// TIA Portal V17 export
// export: Created 2022-03-12T16:05:29.6133544Z, ExportSetting WithDefaults, DisplayName Totally Integrated Automation Portal, DisplayVersion V17, DisplayName TIA Portal Openness, DisplayVersion V17, DisplayName TIA Portal Version Control Interface, DisplayVersion V17, DisplayName STEP 7 Professional, DisplayVersion V17, DisplayName STEP 7 Safety, DisplayVersion V17, DisplayName WinCC Advanced / Unified PC, DisplayVersion V17
DATA_BLOCK "StatusCfg"   // DB31602
TITLE = CPG_StatusCfg
{ S7_Optimized_Access := 'TRUE' }
AUTHOR : tech.team.motioncontrol@siemens.com
FAMILY : CPG
VERSION : 1.0
// Support: tech.team.motioncontrol@siemens.com
// Fax: +49 (0) 9131/98-1297
// stored: AutoNumber true, DBAccessibleFromOPCUA true, DBAccessibleFromWebserver true, IsOnlyStoredInLoadMemory false, IsRetainMemResEnabled false, IsWriteProtectedInAS false, MemoryReserve 0
   VAR
      Event { ExternalAccessible := 'False'; ExternalVisible := 'False'; ExternalWritable := 'False'; S7_SetPoint := 'True'} : Array[0.."CPG_NO_OF_CFG_STATUS_UPPER_LIM"] of "CPG_typeEventCfg";
   END_VAR
BEGIN
   // Event[0] : Status Test
   // Event[1] : 'Alarms Present'
   // Event[2] : 'Waiting for Reset Cmd'
   // Event[3] : 'Waiting for Start Cmd'
   // Event[4] : 'Not Ready for Motion'
   // Event[5] : 'Waiting for No Motion'
   // Event[6] : 'Waiting to start Gearing'
   // Event[7] : 'Waiting to Finish'
   // Event[8] : 'Waiting for Un-Hold Cmd'
   // Event[9] : 'Waiting for Mat. Supply'
   // Event[10] : Spare
   // Event[11] : Spare
   // Event[12] : Spare
   // Event[13] : Spare
   // Event[14] : Spare
   // Event[15] : Spare
   // Event[16] : Spare
   // Event[17] : Spare
   // Event[18] : Spare
   // Event[19] : Spare
   Event[0].ID := 0;
   Event[1].ID := 1;
   Event[2].ID := 2;
   Event[3].ID := 3;
   Event[4].ID := 4;
   Event[5].ID := 5;
   Event[6].ID := 6;
   Event[7].ID := 7;
   Event[8].ID := 8;
   Event[9].ID := 9;
   Event[10].ID := 10;
   Event[11].ID := 11;
   Event[12].ID := 12;
   Event[13].ID := 13;
   Event[14].ID := 14;
   Event[15].ID := 15;
   Event[16].ID := 16;
   Event[17].ID := 17;
   Event[18].ID := 18;
   Event[19].ID := 19;
   Event[0].message[0..1] := 'Status Test';
   Event[0].message[2] := 'Los Status Test';
   Event[1].message[0] := 'Alarms Present';
   Event[1].message[1] := 'Alarme anstehend';
   Event[1].message[2] := 'Las Alarms Present';
   Event[2].message[0] := 'Waiting for Reset PB';
   Event[2].message[1] := 'Warte auf Reset Taste';
   Event[2].message[2] := 'Esperando de Reajustar PB';
   Event[3].message[0] := 'Waiting for Start PB';
   Event[3].message[1] := 'Warten auf Start Taste';
   Event[3].message[2] := 'Esperando de Comenzar PB';
   Event[4].message[0] := 'Not Ready for Motion';
   Event[4].message[1] := 'Maschine nicht anlaufbereit';
   Event[4].message[2] := 'No Listo para Movimiento';
   Event[5].message[0] := 'Waiting for No Motion';
   Event[5].message[1] := 'Warte auf Maschinenstillstand';
   Event[5].message[2] := 'Esperando No Movimiento';
   Event[6].message[0] := 'Waiting to start Gearing';
   Event[6].message[1] := 'Warte auf Start Getriebegleichlauf';
   Event[6].message[2] := 'Waiting to start Gearing';
   Event[7].message[0] := 'Waiting to Finish';
   Event[7].message[1] := 'Warte auf Ende Leerfahren';
   Event[7].message[2] := 'Esperando para Terminar';
   Event[8].message[0] := 'Waiting for Un-Hold PB';
   Event[8].message[1] := 'Warte auf Un-Hold Taste';
   Event[8].message[2] := 'Waiting for Un-Hold PB';
   Event[9].message[0] := 'Waiting for Mat. Supply';
   Event[9].message[1] := 'Warte auf Materialversorgung';
   Event[9].message[2] := 'Waiting for Mat. Supply';
   Event[10].message[0] := 'Spare';
   Event[10].message[1] := 'Reserve';
   Event[10].message[2] := 'Spare';
   Event[11].message[0] := 'Spare';
   Event[11].message[1] := 'Reserve';
   Event[11].message[2] := 'Spare';
   Event[12].message[0] := 'Spare';
   Event[12].message[1] := 'Reserve';
   Event[12].message[2] := 'Spare';
   Event[13].message[0] := 'Spare';
   Event[13].message[1] := 'Reserve';
   Event[13].message[2] := 'Spare';
   Event[14].message[0] := 'Spare';
   Event[14].message[1] := 'Reserve';
   Event[14].message[2] := 'Spare';
   Event[15].message[0] := 'Spare';
   Event[15].message[1] := 'Reserve';
   Event[15].message[2] := 'Spare';
   Event[16].message[0] := 'Spare';
   Event[16].message[1] := 'Reserve';
   Event[16].message[2] := 'Spare';
   Event[17].message[0] := 'Spare';
   Event[17].message[1] := 'Reserve';
   Event[17].message[2] := 'Spare';
   Event[18].message[0] := 'Spare';
   Event[18].message[1] := 'Reserve';
   Event[18].message[2] := 'Spare';
   Event[19].message[0] := 'Spare';
   Event[19].message[1] := 'Reserve';
   Event[19].message[2] := 'Spare';
END_DATA_BLOCK
